FUNCTION_BLOCK FB_ComauInterface
VAR_INPUT
END_VAR
VAR_OUTPUT
END_VAR
VAR
	// Udp related
	{attribute 'tc_no_symbol'}
	udpClient : FB_UdpClient(0, 0, 0, 0, 0, 0, 0);	// Dummy constructor
	{attribute 'tc_no_symbol'}
	rxUdp : ST_RxComau;
	{attribute 'tc_no_symbol'}
	txUdp : ST_TxComau;
END_VAR

// Update udpClient
udpClient();


txUdp.udp_key := 32;
txUdp.beta := 1.0;
txUdp.omega := 1.0;

METHOD FB_exit : BOOL
VAR_INPUT
	bInCopyCode : BOOL; // if TRUE, the exit method is called for exiting an instance that is copied afterwards (online change).
END_VAR
END_METHOD

METHOD FB_init : BOOL
VAR_INPUT
	bInitRetains : BOOL; // if TRUE, the retain variables are initialized (warm start / cold start)
	bInCopyCode : BOOL;  // if TRUE, the instance afterwards gets moved into the copy code (online change)
	
	// Init variables
	remoteIpAddr : UDINT;
	remotePort : UINT;
	localPort : UINT;
END_VAR
// Initilize udpClient
udpClient.FB_init(
	bInitRetains,
	bInCopyCode,
	remoteIpAddr,
	remotePort,
	localPort,
	SIZEOF(rxUdp),
	ADR(rxUdp),
	SIZEOF(txUdp),
	ADR(txUdp)
);
END_METHOD

METHOD FB_reinit : BOOL
VAR_INPUT
END_VAR
END_METHOD

END_FUNCTION_BLOCK

(* stored: Version 1.1.0.1, ProductVersion 3.1.4022.7
   POU FB_ComauInterface: Id {7f6fcfb6-ea5d-4e07-bbf6-5b138a56f61f}, SpecialFunc None
   Method FB_exit: Id {f18839c2-6d63-4a3d-ad66-5f830bcc3ab8}
   Method FB_init: Id {e202aff2-65cb-4030-9293-23617d8046a4}
   Method FB_reinit: Id {09f56272-fe35-4170-800b-7842448d6227} *)
